      # calculate point 201's preheat
      pushtipforward2 = 0.012 - pushtipforward + deepchambumpmm # 12 mm forward to clear the existing extrudant (but still have the extrudant from this extrusion join the existing). subtract from previous to make it constant even if you change pushtipforward1
      preheatdistance = 0.010 # 10 mm . above what it would be pushed down
      point201a = p[p201x, p201y, z + preheatdistance, rx, ry, rz]
      p201bx = p201x + l1delxunit * pushtipforward2
      p201by = p201y + l1delyunit * pushtipforward2
      point201b = p[p201bx, p201by, z + preheatdistance, rx, ry, rz]
      point201c = p[p201bx, p201by, z, rx, ry, rz]

      # calculate point 202
      p202x = p201x + wd3 * l1delxunit
      p202y = p201y + wd3 * l1delyunit
      point202 = p[p202x, p202y, z, rx, ry, rz]

      struct2 = struct(point1=point1, point2=point2, point3=point3, point4=point4, point5=point5, point201=point201, point202=point202, point201a=point201a, point201b=point201b, point201c=point201c, point2a=point2a, point101=point101, point102=point102, point103=point103)
      return struct2
  end

  def calculate_LtAD_points_cover_left(struct1, leftwallthick, rightwallthick, deepcovercham):
      # get the stuff from the struct
      pointintersect = struct1[0]
      x0 = pointintersect[0]
      y0 = pointintersect[1]
      z0 = pointintersect[2]
      heading1 = struct1[1]
      heading2 = struct1[2]
      heading3 = struct1[3]
      l1delxunit = struct1[4]
      l1delyunit = struct1[5]
      l2delxunit = struct1[6]
      l2delyunit = struct1[7]

      # CONST
      welddistance1 = 6 # first path first leg (left side of L)
      welddistance2 = 6 # first path second leg (Right Side of L) # inches
      welddistance3 = 3 # second path (down sidewall) # inches

      wd1 = welddistance1 * 25.4 / 1000
      wd2 = welddistance2 * 25.4 / 1000
      wd3 = welddistance3 * 25.4 / 1000
      leftwallthickmm = leftwallthick * 25.4 / 1000 # in this step corner right, this is distance from left edge
      rightwallthickmm =  rightwallthick * 25.4 / 1000 # in this step corner right, this is distance from right edge

      if deepcovercham:
          deepchambumpmm = 0.09 * 25.4/1000 # if there is a deep chamfer on the cover, bump the welder inwards 0.09 more inches.
      else:
          deepchambumpmm = 0.0
      end

      # first, check if we need a lift column raise
      # (we do, because for maximum reach we want to make the lift pedestal be even with the top of the covers)
      zpi = pointintersect[2]
      if zpi > 0:
          liftcolumnzneeded = zpi * 1000.0 # the robot uses coordinates in meters, but the lift column uses coordinates in mm
          z0 = 0
      else:
          z0 = zpi
      end

      # first and second path

      # calculate rxryrz1 (facing down, preheat rightish)
      # start with rxryrz = 0,0,0 (gun facing up, preheat facing y+ axis)
      # rotate it 180 degrees about x axis. gun facing down, preheat facing y- axis
      # rotate it about 135 degrees ccw about z axis. x+ to heading3 is about 225 degrees. so our angle is heading3 - 90 degrees
      m1 = get_rotation_matrix_from_description("x", -1, 180 * pi / 180) # rotation 1: 180 degrees forward about x axis
      m2 = get_rotation_matrix_from_description("z", 1, heading3 - pi/2) # rotation 2
      m3 = multiply_matrix(m2, m1) #we rotate m1 first then m2, so we multiply in backwards order: 2 then 1
      rxryrz1 = convert_matrix_to_axang(m3)
      rx1 = rxryrz1[0]
      ry1 = rxryrz1[1]
      rz1 = rxryrz1[2]

      # calculate rxryrz2 (gun facing down, preheat facing right and back)
      # rotate 180 degrees about x. then rotate (90 deg + heading1 degrees) about z ccw
      m1 = get_rotation_matrix_from_description("x", -1, 180 * pi / 180)
      m2 = get_rotation_matrix_from_description("z", 1, heading1 + pi/2)
      m3 = multiply_matrix(m2, m1) #we rotate m1 first then m2, so we multiply in backwards order: 2 then 1
      rxryrz2 = convert_matrix_to_axang(m3)
      rx2 = rxryrz2[0]
      ry2 = rxryrz2[1]
      rz2 = rxryrz2[2]

      # calculate point centerchamfers (where the center of the two chamfers intersect
      pcx = x0 + (leftwallthickmm + deepchambumpmm) * l1delxunit + (rightwallthickmm + deepchambumpmm) * l2delxunit
      pcy = y0 + (leftwallthickmm + deepchambumpmm) * l1delyunit + (rightwallthickmm + deepchambumpmm) * l2delyunit
      pcz = z0

      # calculate point1 (start of weld)
      p1x = pcx + l2delxunit * wd1
      p1y = pcy + l2delyunit * wd1
      p1z = pcz
      point1 = p[p1x, p1y, p1z, rx1, ry1, rz1]

      # calculate point2 (end of segment 1)
      p2x = pcx
      p2y = pcy
      p2z = pcz
      point2 = p[p2x, p2y, p2z, rx1, ry1, rz1]

      # calculate point3 (point at end of turn)
      slide = 0.00 # slide distance : the distance the tip slides forward as it turns
      p3x = pcx + slide * l1delxunit
      p3y = pcy + slide * l1delyunit
      p3z = pcz
      point3 = p[p3x, p3y, p3z, rx2, ry2, rz2]

      # calculate point4 (end of segment 2)
      p4x = pcx + wd2 * l1delxunit
      p4y = pcy + wd2 * l1delyunit
      p4z = pcz
      point4 = p[p4x, p4y, p4z, rx2, ry2, rz2]

      # third path

      # calculate rxryrz3 (gun pointing down, preheat pointing toward corner. for left seam, pointing left)
      # start with rxryrz = 0,0,0 (gun facing up, preheat facing y+ axis.
      # rotate it 180 degrees about x axis. gun facing down, preheat facing y- axis
      # rotate it about 45 degrees ccw about z axis. x+ to heading1 is about 135 degrees. so our angle is heading1 - 90 degrees
      m1 = get_rotation_matrix_from_description("x", -1, 180 * pi / 180) # rotation 1: 180 degrees forward about x axis
      m2 = get_rotation_matrix_from_description("z", 1, heading1 - pi/2) # rotation 2
      m3 = multiply_matrix(m2, m1) #we rotate m1 first then m2, so we multiply in backwards order: 2 then 1
      rxryrz3 = convert_matrix_to_axang(m3)
      rx3 = rxryrz3[0]
      ry3 = rxryrz3[1]
      rz3 = rxryrz3[2]

      # calculate rxryrz4 (gun at 45 around corner)
      m1 = get_rotation_matrix_from_description("x", -1, 135 * pi / 180) # rotation 1: 135 degrees forward about x axis
      m2 = get_rotation_matrix_from_description("z", 1, heading1 - pi/2)
      m3 = multiply_matrix(m2, m1) #we rotate m1 first then m2, so we multiply in backwards order: 2 then 1
      rxryrz4 = convert_matrix_to_axang(m3)
      rx4 = rxryrz4[0]
      ry4 = rxryrz4[1]
      rz4 = rxryrz4[2]

      # calculate rxryrz5 (gun straight into left seam side chamfer, preheat down)
      # rotate about x 90 (forward). then rotate about z ~ 45 (ccw)
      m1 = get_rotation_matrix_from_description("x", -1, 90 * pi / 180)
      m2 = get_rotation_matrix_from_description("z", 1, heading1 - pi/2)
      m3 = multiply_matrix(m2, m1) #we rotate m1 first then m2, so we multiply in backwards order: 2 then 1
      rxryrz5 = convert_matrix_to_axang(m3)
      rx5 = rxryrz5[0]
      ry5 = rxryrz5[1]
      rz5 = rxryrz5[2]

      # calculate pointtopcham (the point at the top of the endwall chamfer) ( WHERE POINT3 WOULD BE IF RADIUS WAS 0)
      ptcx = x0 + rightwallthickmm * l2delxunit
      ptcy = y0 + rightwallthickmm * l2delyunit
      ptcz = z0

      # calculate point201 (weld start)
      # if deepchamfer, just ignore that. because if its deep chamfer then it filled more as well. so the hot extrudant should be to the same spot (same distance from the pointtopcham) whether it's big weld or small weld
      adjust = 0.0 # if you want to move the start point further away from corner (positive, mm) or closer to corner
      p201x = x0 + rightwallthickmm * l2delxunit + leftwallthickmm * l1delxunit + adjust * l1delxunit
      p201y = y0 + rightwallthickmm * l2delyunit + leftwallthickmm * l1delyunit + adjust * l1delyunit
      p201z = z0
      point201 = p[p201x, p201y, p201z, rx3, ry3, rz3]

      # the round over distance is the distance from pointbottomvcham to point2 (which will be the same as distance to p4)
      roundoverdistance = 0.05
      rod = roundoverdistance * 25.4 / 1000

      # calculate point202 (start of roundover)
      p202x = ptcx + rod * l1delxunit
      p202y = ptcy + rod * l1delyunit
      p202z = z0
      point202 = p[p202x, p202y, p202z, rx3, ry3, rz3]

      # calculate point203 (middle of roundover)
      # we know that the angle is exactly 90 degrees
      delta = calc_rod_midpoint_90deg(rod)
      p203z = ptcz - delta
      p203x = ptcx + delta * l1delxunit
      p203y = ptcy + delta * l1delyunit
      point203 = p[p203x, p203y, p203z, rx4, ry4, rz4]

      # calculate point204 (end of roundover)
      point204 = p[ptcx, ptcy, ptcz - rod, rx5, ry5, rz5]

      # calculate trail out points (tilt back and ride)
      botvcham = wd3 # where is the bottom of the v chamfer (z distance from top corner)
      tcpdiff = 14 # mm. the difference between backofhole tcp and welder tcp (tip)
      # point101 will still use backofhole, but points 102 and 103 will use normal weld tip tcp
      # calculate point5a (point101) (start of tilt back) (start of unflatten)
      dist = 1.5 * 25.4/1000 + tcpdiff/1000 # distance from botvcham
      p101x = ptcx
      p101y = ptcy
      p101z = ptcz - wd3 + dist
      point101 = p[p101x, p101y, p101z, rx5, ry5, rz5]

      # calculate point5b (point 102) (end of unflatten)
      dist = 0.5 * 25.4 / 1000
      tiltraise = 0.006
      p102x = ptcx + l1delxunit * tiltraise * -1
      p102y = ptcy + l1delyunit * tiltraise * -1
      p102z = ptcz - wd3 + dist

      # calculate rxryrz
      tiltangledeg = 10 # ten degree angle of tilt
      m1 = get_rotation_matrix_from_description("x", -1, (90 + tiltangledeg) * pi / 180) # rotation 1: 135 degrees forward about x axis
      m2 = get_rotation_matrix_from_description("z", 1, heading1 - pi/2)
      m3 = multiply_matrix(m2, m1) #we rotate m1 first then m2, so we multiply in backwards order: 2 then 1
      rxryrz = convert_matrix_to_axang(m3)
      rx = rxryrz[0]
      ry = rxryrz[1]
      rz = rxryrz[2]
      point102 = p[p102x, p102y, p102z, rx, ry, rz]

      # calculate point 5c (point 103) (end of smear)
      dist = -2 * 25.4/1000
      point103 = p[p102x, p102y, ptcz - wd3 + dist, rx, ry, rz]

      # return
      struct2 = struct(point1=point1, point2=point2, point3=point3, point4=point4, point201=point201, point202=point202, point203=point203, point204=point204, point101=point101, point102=point102, point103=point103)
      return struct2


  end

  def calculate_LtAD_points_cover_right(struct1, leftwallthick, rightwallthick, deepcovercham):
      # get the stuff from the struct
      pointintersect = struct1[0]
      x0 = pointintersect[0]
      y0 = pointintersect[1]
      z0 = pointintersect[2]
      heading1 = struct1[1]
      heading2 = struct1[2]
      heading3 = struct1[3]
      l1delxunit = struct1[4]
      l1delyunit = struct1[5]
      l2delxunit = struct1[6]
      l2delyunit = struct1[7]

      # CONST
      welddistance1 = 6 # first path first leg (left side of L)
      welddistance2 = 6 # first path second leg (Right Side of L) # inches
      welddistance3 = 3 # second path (down sidewall) # inches

      wd1 = welddistance1 * 25.4 / 1000
      wd2 = welddistance2 * 25.4 / 1000
      wd3 = welddistance3 * 25.4 / 1000
      leftwallthickmm = leftwallthick * 25.4 / 1000 # in this step corner right, this is distance from left edge
      rightwallthickmm =  rightwallthick * 25.4 / 1000 # in this step corner right, this is distance from right edge

      if deepcovercham:
          deepchambumpmm = 0.09 * 25.4/1000 # if there is a deep chamfer on the cover, bump the welder inwards 0.09 more inches.
      else:
          deepchambumpmm = 0.0
      end

      # first, check if we need a lift column raise
      # (we do, because for maximum reach we want to make the lift pedestal be even with the top of the covers)
      zpi = pointintersect[2]
      if zpi > 0:
          liftcolumnzneeded = zpi * 1000.0 # the robot uses coordinates in meters, but the lift column uses coordinates in mm
          z0 = 0
      else:
          z0 = zpi
      end

      # first and second path

      # calculate rxryrz1 (facing down, preheat rightish)
      # start with rxryrz = 0,0,0 (gun facing up, preheat facing y+ axis)
      # rotate it 180 degrees about x axis. gun facing down, preheat facing y- axis
      # rotate it about 135 degrees ccw about z axis. x+ to heading3 is about 225 degrees. so our angle is heading3 - 90 degrees
      m1 = get_rotation_matrix_from_description("x", -1, 180 * pi / 180) # rotation 1: 180 degrees forward about x axis
      m2 = get_rotation_matrix_from_description("z", 1, heading3 - pi/2) # rotation 2
      m3 = multiply_matrix(m2, m1) #we rotate m1 first then m2, so we multiply in backwards order: 2 then 1
      rxryrz1 = convert_matrix_to_axang(m3)
      rx1 = rxryrz1[0]
      ry1 = rxryrz1[1]
      rz1 = rxryrz1[2]

      # calculate rxryrz2 (gun facing down, preheat facing right and back)
      # rotate 180 degrees about x. then rotate (90 deg + heading1 degrees) about z ccw
      m1 = get_rotation_matrix_from_description("x", -1, 180 * pi / 180)
      m2 = get_rotation_matrix_from_description("z", 1, heading1 + pi/2)
      m3 = multiply_matrix(m2, m1) #we rotate m1 first then m2, so we multiply in backwards order: 2 then 1
      rxryrz2 = convert_matrix_to_axang(m3)
      rx2 = rxryrz2[0]
      ry2 = rxryrz2[1]
      rz2 = rxryrz2[2]

      # calculate point centerchamfers (where the center of the two chamfers intersect
      pcx = x0 + (leftwallthickmm + deepchambumpmm) * l1delxunit + (rightwallthickmm + deepchambumpmm) * l2delxunit
      pcy = y0 + (leftwallthickmm + deepchambumpmm) * l1delyunit + (rightwallthickmm + deepchambumpmm) * l2delyunit
      pcz = z0

      # calculate point1 (start of weld)
      p1x = pcx + l2delxunit * wd1
      p1y = pcy + l2delyunit * wd1
      p1z = pcz
      point1 = p[p1x, p1y, p1z, rx1, ry1, rz1]

      # calculate point2 (end of segment 1)
      p2x = pcx
      p2y = pcy
      p2z = pcz
      point2 = p[p2x, p2y, p2z, rx1, ry1, rz1]

      # calculate point3 (point at end of turn)
      slide = 0.00 # slide distance : the distance the tip slides forward as it turns
      p3x = pcx + slide * l1delxunit
      p3y = pcy + slide * l1delyunit
      p3z = pcz
      point3 = p[p3x, p3y, p3z, rx2, ry2, rz2]

      # calculate point4 (end of segment 2)
      p4x = pcx + wd2 * l1delxunit
      p4y = pcy + wd2 * l1delyunit
      p4z = pcz
      point4 = p[p4x, p4y, p4z, rx2, ry2, rz2]

      # third path

      # calculate rxryrz3 (gun pointing down, preheat pointing toward corner. for right seam, pointing right)
      # start with rxryrz = 0,0,0 (gun facing up, preheat facing y+ axis.
      # rotate it 180 degrees about x axis. gun facing down, preheat facing y- axis
      # rotate it about 135 degrees ccw about z axis. x+ to heading3 is about 225 degrees. so our angle is heading3 - 90 degrees
      m1 = get_rotation_matrix_from_description("x", -1, 180 * pi / 180) # rotation 1: 180 degrees forward about x axis
      m2 = get_rotation_matrix_from_description("z", 1, heading3 - pi/2) # rotation 2
      m3 = multiply_matrix(m2, m1) #we rotate m1 first then m2, so we multiply in backwards order: 2 then 1
      rxryrz3 = convert_matrix_to_axang(m3)
      rx3 = rxryrz3[0]
      ry3 = rxryrz3[1]
      rz3 = rxryrz3[2]

      # calculate rxryrz4 (gun at 45 around corner)
      m1 = get_rotation_matrix_from_description("x", -1, 135 * pi / 180) # rotation 1: 135 degrees forward about x axis
      m2 = get_rotation_matrix_from_description("z", 1, heading3 - pi/2)
      m3 = multiply_matrix(m2, m1) #we rotate m1 first then m2, so we multiply in backwards order: 2 then 1
      rxryrz4 = convert_matrix_to_axang(m3)
      rx4 = rxryrz4[0]
      ry4 = rxryrz4[1]
      rz4 = rxryrz4[2]

      # calculate rxryrz5 (gun straight into right seam side chamfer, preheat down)
      # rotate about x 90 (forward). then rotate about z ~ 135 (ccw)
      m1 = get_rotation_matrix_from_description("x", -1, 90 * pi / 180)
      m2 = get_rotation_matrix_from_description("z", 1, heading3 - pi/2)
      m3 = multiply_matrix(m2, m1) #we rotate m1 first then m2, so we multiply in backwards order: 2 then 1
      rxryrz5 = convert_matrix_to_axang(m3)
      rx5 = rxryrz5[0]
      ry5 = rxryrz5[1]
      rz5 = rxryrz5[2]

      # calculate rxryrz6 (gun straight into right seam side chamfer, preheat down, 10 degrees tiltback)
      tiltangledeg = 10 # ten degree angle of tilt
      m1 = get_rotation_matrix_from_description("x", -1, (90 + tiltangledeg) * pi / 180) # rotation 1: 135 degrees forward about x axis
      m2 = get_rotation_matrix_from_description("z", 1, heading3 - pi/2)
      m3 = multiply_matrix(m2, m1) #we rotate m1 first then m2, so we multiply in backwards order: 2 then 1
      rxryrz6 = convert_matrix_to_axang(m3)
      rx6 = rxryrz6[0]
      ry6 = rxryrz6[1]
      rz6 = rxryrz6[2]

      # calculate pointtopcham (the point at the top of the endwall chamfer) ( WHERE POINT3 WOULD BE IF RADIUS WAS 0)
      ptcx = x0 + leftwallthickmm * l1delxunit
      ptcy = y0 + leftwallthickmm * l1delyunit
      ptcz = z0

      # calculate point201 (weld start)
      # if deepchamfer, just ignore that. because if its deep chamfer then it filled more as well. so the hot extrudant should be to the same spot (same distance from the pointtopcham) whether it's big weld or small weld
      adjust = 0.0 # if you want to move the start point further away from corner (positive, mm) or closer to corner
      p201x = x0 + rightwallthickmm * l2delxunit + leftwallthickmm * l1delxunit + adjust * l2delxunit
      p201y = y0 + rightwallthickmm * l2delyunit + leftwallthickmm * l1delyunit + adjust * l2delyunit
      p201z = z0
      point201 = p[p201x, p201y, p201z, rx3, ry3, rz3]

      # the round over distance is the distance from pointbottomvcham to point2 (which will be the same as distance to p4)
      roundoverdistance = 0.05
      rod = roundoverdistance * 25.4 / 1000

      # calculate point202 (start of roundover)
      p202x = ptcx + rod * l2delxunit
      p202y = ptcy + rod * l2delyunit
      p202z = z0
      point202 = p[p202x, p202y, p202z, rx3, ry3, rz3]

      # calculate point203 (middle of roundover)
      # we know that the angle is exactly 90 degrees
      delta = calc_rod_midpoint_90deg(rod)
      p203z = ptcz - delta
      p203x = ptcx + delta * l2delxunit
      p203y = ptcy + delta * l2delyunit
      point203 = p[p203x, p203y, p203z, rx4, ry4, rz4]

      # calculate point204 (end of roundover)
      point204 = p[ptcx, ptcy, ptcz - rod, rx5, ry5, rz5]

      # calculate trail out points (tilt back and ride)
      botvcham = wd3 # where is the bottom of the v chamfer (z distance from top corner)
      tcpdiff = 14 # mm. the difference between backofhole tcp and welder tcp (tip)
      # point101 will still use backofhole, but points 102 and 103 will use normal weld tip tcp
      # calculate point5a (point101) (start of tilt back) (start of unflatten)
      dist = 1.5 * 25.4/1000 + tcpdiff/1000 # distance from botvcham
      p101x = ptcx
      p101y = ptcy
      p101z = ptcz - wd3 + dist
      point101 = p[p101x, p101y, p101z, rx5, ry5, rz5]

      # calculate point5b (point 102) (end of unflatten)
      dist = 0.5 * 25.4 / 1000
      tiltraise = 0.006
      p102x = ptcx + l2delxunit * tiltraise * -1
      p102y = ptcy + l2delyunit * tiltraise * -1
      p102z = ptcz - wd3 + dist
      point102 = p[p102x, p102y, p102z, rx6, ry6, rz6]

      # calculate point 5c (point 103) (end of smear)
      dist = -2 * 25.4/1000
      point103 = p[p102x, p102y, ptcz - wd3 + dist, rx6, ry6, rz6]

      # return
      struct2 = struct(point1=point1, point2=point2, point3=point3, point4=point4, point201=point201, point202=point202, point203=point203, point204=point204, point101=point101, point102=point102, point103=point103)
      return struct2

  end


  def main_calculate_cover_straight(p11, p12, p21, p22, sidewallthick, leftpoint, rightpoint, deepcovercham):
      struct1 = analyze_touchpoints_only_cover_straight(p11, p12, p21, p22, leftpoint)
      struct2 = calculate_straight_points_cover(struct1, sidewallthick, leftpoint, rightpoint, deepcovercham)
      #struct2 = calculate_DOtA_points_left_extended(struct1, list1, chamferover, chamferup, tcp_pose_top)
      #struct3 = check_validity_left(struct1, struct2)
      return struct2

  end

  # calculates the line of intersection of the sidewall plane (assumed vertical) and the cover plane (assumed perpendicular to sidewall plane)
  # returns a struct containing point0 (point on the intersection line, same y as leftpoint) and 3 components of the unit vector left to right and 2 components of the other direction in 2d
  def analyze_touchpoints_only_cover_straight(p11, p12, p21, p22, leftpoint):
      # calculate slope of sidewall in x-y plane
      # get the raw points from the first line
      l1p1x=p11[0]
      l1p1y=p11[1]
      l1p2x=p12[0]
      l1p2y=p12[1]

      # equate the first line in 2d space
      ml1 = (l1p2y-l1p1y) / (l1p2x-l1p1x)

      # b = y - mx
      bl1 = l1p1y - ml1 * l1p1x

      # calculate the cover plane
      # if two planes are perpendicular, then their normal vectors must be perpendicular.
      # the first planes normal vector is n1, which is taken from the equation of the plane ax + by + cz = d -> <a, b, c>
      # the second plane's normal vector is perpendicular to all vectors contained in the plane
      # p21 to p22 is a vector v contained within plane 2.
      # n2 is normal to both n1 AND v. to achieve a vector that is normal to both, take the cross product

      # plane 1 (y = mx + b) -> (b = -mx +1y +0z)
      n1 = [-1 * ml1, 1, 0]

      # v=P2−P1=(x2−x1,y2−y1,z2−z1)
      v = [p21[0]-p22[0], p21[1]-p22[1], p21[2]-p22[2]]

      #v n2 = cross product of n1 and v
      n2x = n1[1]*v[2] - n1[2]*v[1]
      n2y = n1[2]*v[0] - n1[0]*v[2]
      n2z = n1[0]*v[1] - n1[1]*v[0]
      n2 = [n2x, n2y, n2z]

      # find the d of the second plane
      # n2x * x + n2y * y + n2z * z = d0
      d = n2x * p21[0] + n2y * p21[1] + n2z * p21[2]

      # find the intersection line of the two planes
      # find the direction vector of that line by taking the cross product of the normal vector of those two planes
      v3x = n1[1]*n2[2] - n1[2]*n2[1]
      v3y = n1[2]*n2[0] - n1[0]*n2[2]
      v3z = n1[0]*n2[1] - n1[1]*n2[0]
      v3 = [v3x, v3y, v3z]

      # normalize the vector so the magnitude is 1
      magnitude2 = v3x * v3x + v3y * v3y + v3z * v3z
      magnitude = sqrt(magnitude2)
      v3xunit = v3x/magnitude
      v3yunit = v3y/magnitude
      v3zunit = v3z/magnitude

      # make sure it is going the right way (from left to right). make sure the v3yunit is positive
      if v3yunit < 0:
          v3xunit = v3xunit * -1
          v3yunit = v3yunit * -1
          v3zunit = v3zunit * -1
      end

      # next we have to find a point on the line by setting one of the dimensions and solving the system of equations
      # i will pick the y value of the left teach point
      y = leftpoint[1]
      # plane 1: -ml1 * x + 1 * y + 0 * z = bl1
      # -ml1 * x = bl1 - y
      x = (bl1 - y)/ (-1 * ml1)
      # plane 2: d = n2x * x + n2y * y + n2z * z
      # (d - n2x * x - n2y * y) = n2z * z
      z = (d - n2x * x - n2y * y) / n2z

      # make point0 into a pose
      point0 = p[x, y, z, 0, 0, 0]

      # find heading of main line
      heading1 = convert_uv_to_heading(v3xunit, v3yunit)

      # make a unit vector perpendicular to this one in the xy plane pointing x -. will be used to move over the chamfer distance
      ml2 = -1 / ml1
      # y = ml2 * x + unknownB
      # vector = [1, ml2]
      mag2 = 1 + ml2 * ml2
      mag = sqrt(mag2)
      v4xunit = 1 / mag
      v4yunit = ml2 / mag
      # switch is to the x direction is negative
      v4xunit = -1 * v4xunit
      v4yunit = -1 * v4yunit

      ret = struct(point0=point0, v3xunit=v3xunit, v3yunit=v3yunit, v3zunit=v3zunit, heading1=heading1, v4xunit=v4xunit, v4yunit=v4yunit)
      return ret
  end

  def calculate_straight_points_cover(struct1, sidewallthick, leftpointteach, rightpointteach, deepcovercham):
      # get the stuff
      point0 = struct1[0]
      p0x = point0[0]
      p0y = point0[1]
      p0z = point0[2]
      v3xunit = struct1[1]
      v3yunit = struct1[2]
      v3zunit = struct1[3]
      heading1 = struct1[4]
      v4xunit = struct1[5]
      v4yunit = struct1[6]
      sidewallthick = sidewallthick
      lpy = leftpointteach[1]
      rpy = rightpointteach[1]

      # first, check if we need a lift column raise
      # (we do, because for maximum reach we want to make the lift pedestal be even with the top of the covers)
      zpi = p0z
      if zpi > 0:
          liftcolumnzneeded = zpi * 1000.0 # the robot uses coordinates in meters, but the lift column uses coordinates in mm
          coverz = 0
      else:
          coverz = zpi
      end

      if deepcovercham:
          deepchambumpmm = 0.09 * 25.4/1000 # if there is a deep chamfer on the cover, bump the welder inwards 0.09 more inches.
      else:
          deepchambumpmm = 0.0
      end

      # calculate pointtopvcham
      chamferover = sidewallthick * 25.4 / 1000.0 + deepchambumpmm
      tiltraise = 0.006 # 6 mm raise needed for the tip to clear the plane during tiltback
      x = p0x + v4xunit * chamferover
      y = p0y + v4yunit * chamferover
      z = coverz + tiltraise

      # calculate rxryrz for tilted back
      # 3 rotations to make this happen.
      # start point is straight up with the preheat pointed in the +y direction.
      # first rotation is 180 degrees about x direction. gun is now pointing straight down with preheat facing -y direction
      m1 = get_rotation_matrix_from_description("x", 1, 180 * pi / 180)
      # second rotation is a 10 degree turn about the x axis (negative direction)
      m2 = get_rotation_matrix_from_description("x", -1, 10 * pi / 180)
      # third rotation is about 180 degrees about the z axis. starting from the -y axis, go until you get to heading1. that will equal heading1 plus 90 degrees
      m3 = get_rotation_matrix_from_description("z", 1, pi/2 + heading1)
      # combine them by multiplying m3 * m2 * m1
      # matrix multiplication is not commutative but it IS associative, so you can do this whichever order
      m4 = multiply_matrix(m2, m1)
      m5 = multiply_matrix(m3, m4)
      rxryrzt = convert_matrix_to_axang(m5)
      rxt = rxryrzt[0]
      ryt = rxryrzt[1]
      rzt = rxryrzt[2]
      pointtopvcham = p[x, y, z, rxt, ryt, rzt]

      # calculate point1 (preheat)
      dist = -1 * 25.4 / 1000.0 # move back 1 inch from
      p1x = x + dist * v3xunit
      p1y = y + dist * v3yunit
      p1z = z + dist * v3zunit
      point1 = p[p1x, p1y, p1z, rxt, ryt, rzt]

      # calculate point2 (start of flatten)
      dist = 0.5 * 25.4 / 1000.0  # half an inch past the top of v chamfer
      p2x = x + dist * v3xunit
      p2y = y + dist * v3yunit
      p2z = z + dist * v3zunit
      point2 = p[p2x, p2y, p2z, rxt, ryt, rzt]

      # calculate rxryrz for nontilted
      # first rotation is 180 degrees about x direction. gun is now pointing straight down with preheat facing -y direction
      m1 = get_rotation_matrix_from_description("x", 1, 180 * pi / 180)
      # third rotation is about 180 degrees about the z axis. starting from the -y axis, go until you get to heading1. that will equal heading1 plus 90 degrees
      m3 = get_rotation_matrix_from_description("z", 1, pi/2 + heading1)
      m5 = multiply_matrix(m3, m1)
      rxryrz = convert_matrix_to_axang(m5)
      rx = rxryrz[0]
      ry = rxryrz[1]
      rz = rxryrz[2]

      # calculate point3 (end of flatten)
      dist = 1.5 * 25.4 / 1000.0  # 1.5 inches past top of v chamfer
      p3x = x + dist * v3xunit
      p3y = y + dist * v3yunit
      p3z = coverz + dist * v3zunit
      point3 = p[p3x, p3y, p3z, rx, ry, rz]

      # calculate distance between leftpoint and rightpoint
      # we have the y distance. we need to find the total distance.
      # the unit vector (v3) should have a magnitude of 1. that's what analyze_touchpoints_only_cover_straight() calculated.
      # so the total distance is y distance * 1 / v3yunit
      ydist = rpy - lpy
      totdist = ydist / v3yunit

      # calculate pointtopvcham2
      x2 = x + v3xunit * totdist
      y2 = y + v3yunit * totdist
      z2 = z + v3zunit * totdist

      # calculate point4 (start of unflatten)
      dist = -1.5 * 25.4 / 1000.0
      p4x = x2 + v3xunit * dist
      p4y = y2 + v3yunit * dist
      p4z = z2 + v3zunit * dist - tiltraise
      point4 = p[p4x, p4y, p4z, rx, ry, rz]

      # calculate point5 (end of unflatten)
      dist = -0.5 * 25.4 / 1000.0
      p5x = x2 + v3xunit * dist
      p5y = y2 + v3yunit * dist
      p5z = z2 + v3zunit * dist
      point5 = p[p5x, p5y, p5z, rxt, ryt, rzt]

      # calculate point6 (end of smear)
      dist = 2 * 25.4 / 1000.0
      p6x = x2 + v3xunit * dist
      p6y = y2 + v3yunit * dist
      p6z = z2 + v3zunit * dist
      point6 = p[p6x, p6y, p6z, rxt, ryt, rzt]


      # return struct
      ret = struct(pointtopvcham=pointtopvcham, point1=point1, point2=point2, point3=point3, point4=point4, point5=point5, point6=point6)
      return ret


  end

  def main_calculate_floor_straight(p11, p12, p21, p22, floorthick, leftpoint, rightpoint):
      struct1 = analyze_touchpoints_only_cover_straight(p11, p12, p21, p22, leftpoint)
      struct2 = calculate_straight_points_floor(struct1, floorthick, leftpoint, rightpoint)
      #struct2 = calculate_DOtA_points_left_extended(struct1, list1, chamferover, chamferup, tcp_pose_top)
      #struct3 = check_validity_left(struct1, struct2)
      return struct2

  end

  # the path for welding a floor straight weld with v chisels on both sides.
  # start at the right side and move left.
  def calculate_straight_points_floor(struct1, floorthick, leftpointteach, rightpointteach):
      # get the stuff
      point0 = struct1[0]
      p0x = point0[0]
      p0y = point0[1]
      p0z = point0[2]
      v3xunit = struct1[1]
      v3yunit = struct1[2]
      v3zunit = struct1[3]
      heading1 = struct1[4]
      v4xunit = struct1[5]
      v4yunit = struct1[6]
      lpy = leftpointteach[1]
      rpy = rightpointteach[1]

      # first, check if we need a lift column raise
      # (we do not, because the floors are low)
      zpi = p0z
      floorz = zpi

      # calculate pointtopvcham (left point) (tilted and tiltraised)
      chamferup = floorthick * 25.4 / 1000.0
      tiltraise = 0.006 # 6 mm raise needed for the tip to clear the plane during tiltback
      # on this one, move the tiltraise distance sideways (towards robot) and the chamferover distance up
      x = p0x + v4xunit * tiltraise * -1
      y = p0y + v4yunit * tiltraise * -1
      z = floorz + chamferup

      # calculate rxryrz for tilted back
      # 3 rotations to make this happen.
      # start point is straight up with the preheat pointed in the +y direction.
      # first rotation is 90 degrees about y axis. positive direction. gun is now pointing in the x+ direction with preheat facing +y direction
      m1 = get_rotation_matrix_from_description("y", 1, 90 * pi / 180)
      # second rotation is about 180 degrees about the z axis. heading1 plus 90 degrees. gun is now pointing directly into the sidewall
      m2 = get_rotation_matrix_from_description("z", 1, pi/2 + heading1)
      # third rotation is 10 degrees about the z axis. gun is now tilted back 10 degrees from the sidewall
      m3 = get_rotation_matrix_from_description("z", 1, 10 * pi / 180)
      # combine them by multiplying m3 * m2 * m1
      # matrix multiplication is not commutative but it IS associative, so you can do this whichever order
      m4 = multiply_matrix(m2, m1)
      m5 = multiply_matrix(m3, m4)
      rxryrzt = convert_matrix_to_axang(m5)
      rxt = rxryrzt[0]
      ryt = rxryrzt[1]
      rzt = rxryrzt[2]
      # the non tilted angle is just m4
      rxryrz = convert_matrix_to_axang(m4)
      rx = rxryrz[0]
      ry = rxryrz[1]
      rz = rxryrz[2]
      pointtopvcham = p[x, y, z, rxt, ryt, rzt]

      # calculate distance between leftpoint and rightpoint
      # we have the y distance. we need to find the total distance.
      # the unit vector (v3) should have a magnitude of 1. that's what analyze_touchpoints_only_cover_straight() calculated.
      # so the total distance is y distance * 1 / v3yunit
      ydist = rpy - lpy
      totdist = ydist / v3yunit

      # calculate pointtopvcham2 (right point) (tilted and tiltraised)
      x2 = x + v3xunit * totdist
      y2 = y + v3yunit * totdist
      z2 = z + v3zunit * totdist
      pointtopvcham2 = p[x2, y2, z2, rxt, ryt, rzt]

      # calculate point1 (preheat)
      dist = 1 * 25.4 / 1000.0 # move back 1 inch from ptvc2 (in this case back means positive)
      p1x = x2 + dist * v3xunit
      p1y = y2 + dist * v3yunit
      p1z = z2 + dist * v3zunit
      point1 = p[p1x, p1y, p1z, rxt, ryt, rzt]

      # calculate point2 (start of flatten)
      dist = -0.5 * 25.4 / 1000.0  # half an inch past the top of v chamfer
      p2x = x2 + dist * v3xunit
      p2y = y2 + dist * v3yunit
      p2z = z2 + dist * v3zunit
      point2 = p[p2x, p2y, p2z, rxt, ryt, rzt]

      # calculate point3 (end of flatten)
      dist = -1.5 * 25.4 / 1000.0  # 1.5 inches past top of v chamfer
      p3x = x2 + dist * v3xunit + tiltraise * v4xunit
      p3y = y2 + dist * v3yunit + tiltraise * v4yunit
      p3z = z2 + dist * v3zunit
      point3 = p[p3x, p3y, p3z, rx, ry, rz]

      # calculate point4 (start of unflatten)
      dist = 1.5 * 25.4 / 1000.0
      p4x = x + v3xunit * dist + tiltraise * v4xunit
      p4y = y + v3yunit * dist + tiltraise * v4yunit
      p4z = z + v3zunit * dist
      point4 = p[p4x, p4y, p4z, rx, ry, rz]

      # calculate point5 (end of unflatten)
      dist = 0.5 * 25.4 / 1000.0
      p5x = x + v3xunit * dist
      p5y = y + v3yunit * dist
      p5z = z + v3zunit * dist
      point5 = p[p5x, p5y, p5z, rxt, ryt, rzt]

      # calculate point6 (end of smear)
      dist = -2 * 25.4 / 1000.0
      p6x = x + v3xunit * dist
      p6y = y + v3yunit * dist
      p6z = z + v3zunit * dist
      point6 = p[p6x, p6y, p6z, rxt, ryt, rzt]

      # return struct
      ret = struct(pointtopvcham=pointtopvcham, point1=point1, point2=point2, point3=point3, point4=point4, point5=point5, point6=point6)
      return ret

  end

  # this function determines the starting touchpoints for homing in on cover lt geometry
  # includes two points above the cover lt, closer to the robot than the lt, facing down
  def get_coverlt_homing_pathpoints(leftpoint, rightpoint):
      # get the teach position points
      lpx = leftpoint[0]
      lpy = leftpoint[1]
      lpz = leftpoint[2]
      rpx = rightpoint[0]
      rpy = rightpoint[1]
      rpz = rightpoint[2]

      # specify the distances from (in meters)
      d0 = 0.05 # how far from the cover to approach from
      d1 = 0.03 # how far the touchpints are pushed closer to the robot
      d2 = 0.00 # how far inwards the touchpoints are pushed

      # rxryrz
      rxryrz = [0.334, 3.124, 0]
      rx = rxryrz[0]
      ry = rxryrz[1]
      rz = rxryrz[2]

      # calculate the points
      ph1 = p[lpx + d1, lpy + d2, lpz + d0, rx, ry, rz] # left side approach
      ph2 = p[rpx + d1, rpy - d2, rpz + d0, rx, ry, rz] # right side approach

      ret = struct(ph1=ph1, ph2=ph2)
      is_robot_at_reachable_spot(leftpoint, ret)
      return ret
  end

  def main_calculate_cover_lt(p11, p12, leftpoint, rightpoint):
      struct1 = analyze_touchpoints_only_cover_lt(p11, p12, leftpoint, rightpoint)
      struct2 = calculate_points_cover_lt(struct1)
      #struct2 = calculate_DOtA_points_left_extended(struct1, list1, chamferover, chamferup, tcp_pose_top)
      #struct3 = check_validity_left(struct1, struct2)
      return struct2

  end

  def analyze_touchpoints_only_cover_lt(p11, p12, leftpoint, rightpoint):
      # calculate the slope of the groove in xy plane
      l1p1x = leftpoint[0]
      l1p1y = leftpoint[1]
      l1p2x = rightpoint[0]
      l1p2y = rightpoint[1]

      # equate the first line in 2d space
      ml1 = (l1p2y-l1p1y) / (l1p2x-l1p1x)

      # b = y - mx
      bl1 = l1p1y - ml1 * l1p1x

      # zraise (how much the z value changes from left point to right point
      zraise = p12[2] - p11[2]

      #get the calcpoints
      leftcalcpoint = [leftpoint[0], leftpoint[1], p11[2]]
      rightcalcpoint = [rightpoint[0], rightpoint[1], p12[2]]
      # get the vector from a to b
      vec = [rightcalcpoint[0] - leftcalcpoint[0], rightcalcpoint[1] - leftcalcpoint[1], rightcalcpoint[2] - leftcalcpoint[2]]
      # get the unit vector in 3d
      mag3d = sqrt(vec[0]*vec[0]+vec[1]*vec[1]+vec[2]*vec[2])
      vec3dunit = [vec[0]/mag3d, vec[1]/mag3d, vec[2]/mag3d]
      # get the unit vector in 2d
      mag2d = sqrt(vec[0]*vec[0]+vec[1]*vec[1])
      vec2dunit = [vec[0]/mag2d, vec[1]/mag2d]
      # get the heading
      heading1 = convert_uv_to_heading(vec2dunit[0], vec2dunit[1])

      ret = struct(leftcalcpoint=leftcalcpoint, rightcalcpoint=rightcalcpoint, vxunit=vec3dunit[0], vyunit=vec3dunit[1], vzunit=vec3dunit[2], heading1=heading1)
      return ret
  end

  def calculate_points_cover_lt(struct1):
      # get the stuff from struct
      leftcalcpoint = struct1[0]
      x = leftcalcpoint[0]
      y = leftcalcpoint[1]
      z = leftcalcpoint[2]
      rightcalcpoint = struct1[1]
      x2 = rightcalcpoint[0]
      y2 = rightcalcpoint[1]
      z2 = rightcalcpoint[2]
      v3xunit = struct1[2]
      v3yunit = struct1[3]
      v3zunit = struct1[4]
      heading1 = struct1[5]

      # first calculate rxryrz f normal and tiltback
      # calculate rxryrz for tilted back
      # 3 rotations to make this happen.
      # start point is straight up with the preheat pointed in the +y direction.
      # first rotation is 180 degrees about x direction. gun is now pointing straight down with preheat facing -y direction
      m1 = get_rotation_matrix_from_description("x", 1, 180 * pi / 180)
      # second rotation is a 10 degree turn about the x axis (negative direction)
      m2 = get_rotation_matrix_from_description("x", -1, 10 * pi / 180)
      # third rotation is about 180 degrees about the z axis. starting from the -y axis, go until you get to heading1. that will equal heading1 plus 90 degrees
      m3 = get_rotation_matrix_from_description("z", 1, pi/2 + heading1)
      # combine them by multiplying m3 * m2 * m1
      # matrix multiplication is not commutative but it IS associative, so you can do this whichever order
      m4 = multiply_matrix(m2, m1)
      m5 = multiply_matrix(m3, m4)
      rxryrzt = convert_matrix_to_axang(m5)
      rxt = rxryrzt[0]
      ryt = rxryrzt[1]
      rzt = rxryrzt[2]

      # calculate rxryrz for nontilted
      # first rotation is 180 degrees about x direction. gun is now pointing straight down with preheat facing -y direction
      m1 = get_rotation_matrix_from_description("x", 1, 180 * pi / 180)
      # third rotation is about 180 degrees about the z axis. starting from the -y axis, go until you get to heading1. that will equal heading1 plus 90 degrees
      m3 = get_rotation_matrix_from_description("z", 1, pi/2 + heading1)
      m5 = multiply_matrix(m3, m1)
      rxryrz = convert_matrix_to_axang(m5)
      rx = rxryrz[0]
      ry = rxryrz[1]
      rz = rxryrz[2]

      tiltraise = 0.006 # 6 mm raise needed for the tip to clear the plane during tiltback

      # calculate points 1-3
      # calculate point1 (preheat)
      dist = -1 * 25.4 / 1000.0 # move back 1 inch from
      p1x = x + dist * v3xunit
      p1y = y + dist * v3yunit
      p1z = z + dist * v3zunit + tiltraise
      point1 = p[p1x, p1y, p1z, rxt, ryt, rzt]

      # calculate point2 (start of flatten)
      dist = 0.5 * 25.4 / 1000.0  # half an inch past the top of v chamfer
      p2x = x + dist * v3xunit
      p2y = y + dist * v3yunit
      p2z = z + dist * v3zunit + tiltraise
      point2 = p[p2x, p2y, p2z, rxt, ryt, rzt]

      # calculate point3 (end of flatten)
      dist = 1.5 * 25.4 / 1000.0  # 1.5 inches past top of v chamfer
      p3x = x + dist * v3xunit
      p3y = y + dist * v3yunit
      p3z = z + dist * v3zunit
      point3 = p[p3x, p3y, p3z, rx, ry, rz]

      # calculate points 4-6
      # calculate point4 (start of unflatten)
      dist = -1.5 * 25.4 / 1000.0
      p4x = x2 + v3xunit * dist
      p4y = y2 + v3yunit * dist
      p4z = z2 + v3zunit * dist
      point4 = p[p4x, p4y, p4z, rx, ry, rz]

      # calculate point5 (end of unflatten)
      dist = -0.5 * 25.4 / 1000.0
      p5x = x2 + v3xunit * dist
      p5y = y2 + v3yunit * dist
      p5z = z2 + v3zunit * dist + tiltraise
      point5 = p[p5x, p5y, p5z, rxt, ryt, rzt]

      # calculate point6 (end of smear)
      dist = 2 * 25.4 / 1000.0
      p6x = x2 + v3xunit * dist
      p6y = y2 + v3yunit * dist
      p6z = z2 + v3zunit * dist + tiltraise
      point6 = p[p6x, p6y, p6z, rxt, ryt, rzt]

      # return struct
      ret = struct(pointtopvcham=leftcalcpoint, point1=point1, point2=point2, point3=point3, point4=point4, point5=point5, point6=point6)
      return ret

  end

  def main_calculate_sleeve_fillet(p1, p2, p3):
      struct1 = analyze_touchpoints_only_sleeve_fillet(p1, p2, p3)
      struct2 = calculate_points_sleeve_fillet(struct1)
      return struct2
  end

  # given 3 points at the intersection of the sleeve and the sidewall, this calculates and returns 3 things:
  # the centerpoint of the circle on the plane, the normal vector of the plane, and the radius of the circle
  # then it returns 4 more things after converting to a vertical circle/plane: heading1 (into the plane), vecn, vecr, vecu
  def analyze_touchpoints_only_sleeve_fillet(p1, p2, p3):
      x1 = p1[0]
      y1 = p1[1]
      z1 = p1[2]
      x2 = p2[0]
      y2 = p2[1]
      z2 = p2[2]
      x3 = p3[0]
      y3 = p3[1]
      z3 = p3[2]

      # calculate plane
      # calculate ab (1->2) vector
      abvec = [x2-x1, y2-y1, z2-z1]
      # calculate ac (1->3) vector
      acvec = [x3-x1, y3-y1, z3-z1]
      #calculate the plane's normal vector = ab x ac

      n = crossproduct(abvec, acvec)
      mag = sqrt(n[0]*n[0]+n[1]*n[1]+n[2]*n[2])
      n = [n[0]/mag, n[1]/mag, n[2]/mag]
      d = n[0] * x1 + n[1] * y1 + n[2] * z1

      # find the circle
      # Midpoint of AB:
      mab = [(x1 + x2)/2, (y1 + y2)/2, (z1 + z2)/2]
      # midpoint of ac
      mac = [(x3 + x1)/2, (y3 + y1)/2, (z3 + z1)/2]
      # Get Normal Vectors to AB and AC in the Plane
      # nab (normal to ab) = abvec x n
      nab = crossproduct(abvec, n)
      # nac (normal to ac) = acvec x n
      nac = crossproduct(acvec, n)
      # Define Perpendicular Bisector Lines
      # Each line goes through a midpoint and extends in the direction of the na_
      # we already have the equations of those lines in point vector form with l1 = mab + s * nab, and l2 = mac + t * nac
      # define all the terms so the math is simpler when i have to do math
      mabx = mab[0]
      maby = mab[1]
      mabz = mab[2]
      nabx = nab[0]
      naby = nab[1]
      nabz = nab[2]
      macx = mac[0]
      macy = mac[1]
      macz = mac[2]
      nacx = nac[0]
      nacy = nac[1]
      nacz = nac[2]
      # find the intersection point using the y and z equations
      # maby + s * naby = macy + t * nacy
      # mabz + s * nabz = macz + t * nacz
      # first solve for s and take
      # t = (macz*naby + maby*nabz - mabz*naby - macy*nabz) / (nacy*nabz - naby*nacz)
      t = (macz*naby + maby*nabz - mabz*naby - macy*nabz) / (nacy*nabz - naby*nacz)
      # s = (t*nacz + macz - mabz) / nabz
      s = (t*nacz + macz - mabz) / nabz
      # find the point
      # pcenter = mac + t * nac
      pcenterx = macx + t * nacx
      pcentery = macy + t * nacy
      pcenterz = macz + t * nacz
      rxryrz = [0.528, 4.631, 0.258] # demo point of the welder pointing forward into a sleeve
      pcenter = p[pcenterx, pcentery, pcenterz, rxryrz[0], rxryrz[1], rxryrz[2]]
      radius = distance_between(pcenterx, pcentery, pcenterz, x1, y1, z1)

      # ------ start calculation of vertical assumption -----
      # assume the plane close to vertical
      # fix it to make it actually vertical
      # calculate the unit vector of up, and the unit vector of right.
      # calculate the heading from the +x axis to pointing straight into the wall.
      # the unit vector of up is [0, 0, 1] (because the plane is verticalized) (for easier calculations)
      # first calculate the normal vector INTO the sidewall (make sure x is negative) and make it a unit vector
      vecn = [n[0], n[1], 0] # vector normal
      if vecn[0] > 0:
          vecn = [-n[0], -n[1], 0]
      end
      mag = sqrt(vecn[0]*vecn[0]+vecn[1]*vecn[1])
      vecn = [vecn[0]/mag, vecn[1]/mag, 0]
      # next calculate the right normal vector (the vector IN the plane that goes to the right)
      vecr = [vecn[1], -1*vecn[0], 0]
      vecu = [0, 0, 1] # vector up
      heading1 = convert_uv_to_heading(vecn[0], vecn[1])


      ret = struct(pcenter=pcenter, planenormalvec=n, radius=radius, heading1=heading1, vecn=vecn, vecr=vecr, vecu=vecu)
      return ret
  end

  def crossproduct(vec1, vec2):
      nx = vec1[1]*vec2[2] - vec1[2]*vec2[1]
      ny = vec1[2]*vec2[0] - vec1[0]*vec2[2]
      nz = vec1[0]*vec2[1] - vec1[1]*vec2[0]
      ret = [nx, ny, nz]
      return ret
  end

  # this function calculates only the four points of the quadrants, for the not real program.
  # these calculations are easier so that's why i'm starting with them first.
  # this assumes a vertical plane
  def calculate_points_sleeve_fillet_quadonly(struct1):
      # get the stuff from the struct
      pcenter = struct1[0]
      pcx = pcenter[0]
      pcy = pcenter[1]
      pcz = pcenter[2]
      planenormalvec = struct1[1]
      radius = struct1[2]
      heading1 = struct1[3]
      vecn = struct1[4]
      vecnx = vecn[0]
      vecny = vecn[1]
      vecr = struct1[5]
      vecrx = vecr[0]
      vecry = vecr[1]
      vecu = struct1[6]
      vecuz = vecu[2]

      # define cushions (the backofhole can't actually touch the intersection of pipe and wall, it travels a certain distance around it
      cushout = 0.006 # 5mm # the cushion out from the wall
      cusharound = 0.006 # 5mm # the cushion around the sleeve.

      # get the top point (point1)
      # take the center point and move up the radius plus the cushions
      p1x = pcx + vecnx * -1 * cushout
      p1y = pcy + vecny * -1 * cushout
      p1z = pcz + vecuz * radius + vecuz * cusharound

      # find rxryrz1
      # first rotation is 135 degrees about the y- direction. 90 degrees to get flat. Tip pointing x-, preheat pointing y+. 45 more degrees to get at that above angle
      m1 = get_rotation_matrix_from_description("y", -1, 135 * pi / 180)
      # second rotation is heading1 – 180 degrees about the z+ axis to get pointing straight into wall. Heading1 should be about 180 degrees
      m2 = get_rotation_matrix_from_description("z", 1, heading1 - 180 * pi/180)
      # combine them by multiplying
      m3 = multiply_matrix(m2, m1)
      rxryrz1 = convert_matrix_to_axang(m3)
      rx1 = rxryrz1[0]
      ry1 = rxryrz1[1]
      rz1 = rxryrz1[2]

      point1 = p[p1x, p1y, p1z, rx1, ry1, rz1]

      # get second point (right) (point2)
      # take the center point and move right the radius plus the cushions
      p2x = pcx + vecrx * radius + vecrx * cusharound + vecnx * -1 * cushout
      p2y = pcy + vecry * radius + vecry * cusharound + vecny * -1 * cushout
      p2z = pcz

      # find rxryrz2
      # first rotation is 90 degrees about the x- axis
      m1 = get_rotation_matrix_from_description("x", -1, 90 * pi / 180)
      # second rotation is About 135 degrees about the z+ axis. This calculation is heading1 – 45 degrees
      m2 = get_rotation_matrix_from_description("z", 1, heading1 - 45 * pi/180)
      # combine them by multiplying
      m3 = multiply_matrix(m2, m1)
      rxryrz2 = convert_matrix_to_axang(m3)
      rx2 = rxryrz2[0]
      ry2 = rxryrz2[1]
      rz2 = rxryrz2[2]

      point2 = p[p2x, p2y, p2z, rx2, ry2, rz2]

      # get the third point (bottom) (point3)
      p3x = pcx + vecnx * -1 * cushout
      p3y = pcy + vecny * -1 * cushout
      p3z = pcz - vecuz * radius - vecuz * cusharound

      # find rxryrz3
      # first rotation is 45 degrees about the y+ axis
      m1 = get_rotation_matrix_from_description("y", 1, 45 * pi / 180)
      # second rotation is About 180 degrees about the z+ axis. This calculation is heading1 degrees
      m2 = get_rotation_matrix_from_description("z", 1, heading1)
      # combine them by multiplying
      m3 = multiply_matrix(m2, m1)
      rxryrz3 = convert_matrix_to_axang(m3)
      rx3 = rxryrz3[0]
      ry3 = rxryrz3[1]
      rz3 = rxryrz3[2]

      point3 = p[p3x, p3y, p3z, rx3, ry3, rz3]

      # get the fourth point (left) (point4)
      p4x = pcx - vecrx * radius - vecrx * cusharound + vecnx * -1 * cushout
      p4y = pcy - vecry * radius - vecry * cusharound + vecny * -1 * cushout
      p4z = pcz

      # find rxryrz4
      # first rotation is 90 degrees about the x+ axis
      m1 = get_rotation_matrix_from_description("x", 1, 90 * pi / 180)
      # second rotation is heading1 + 45 degrees about the z+ axis. approx 225 degrees ccw
      m2 = get_rotation_matrix_from_description("z", 1, heading1 + 45 * pi/180)
      # combine them by multiplying
      m3 = multiply_matrix(m2, m1)
      rxryrz4 = convert_matrix_to_axang(m3)
      rx4 = rxryrz4[0]
      ry4 = rxryrz4[1]
      rz4 = rxryrz4[2]

      point4 = p[p4x, p4y, p4z, rx4, ry4, rz4]

      # return the points
      ret = struct(point1=point1, point2=point2, point3=point3, point4=point4)
      return ret

  end

  # this function calculates the points necessary for the fillet sleeve weld path.
  # this assumes a vertical plane
  def calculate_points_sleeve_fillet(struct1):
      # get the stuff from the struct
      pcenter = struct1[0]
      pcx = pcenter[0]
      pcy = pcenter[1]
      pcz = pcenter[2]
      planenormalvec = struct1[1]
      radius = struct1[2]
      heading1 = struct1[3]
      vecn = struct1[4]
      vecnx = vecn[0]
      vecny = vecn[1]
      vecr = struct1[5]
      vecrx = vecr[0]
      vecry = vecr[1]
      vecu = struct1[6]
      vecuz = vecu[2]

      # define cushions (the backofhole can't actually touch the intersection of pipe and wall, it travels a certain distance around it
      cushout = 0.006 # 5mm # the cushion out from the wall
      cusharound = 0.004 # 5mm # the cushion around the sleeve.

      # get the top point (point1)
      # take the center point and move up the radius plus the cushions
      p1x = pcx + vecnx * -1 * cushout
      p1y = pcy + vecny * -1 * cushout
      p1z = pcz + vecuz * radius + vecuz * cusharound

      # find rxryrz1
      # first rotation is 135 degrees about the y- direction. 90 degrees to get flat. Tip pointing x-, preheat pointing y+. 45 more degrees to get at that above angle
      m1 = get_rotation_matrix_from_description("y", -1, 135 * pi / 180)
      # second rotation is heading1 – 180 degrees about the z+ axis to get pointing straight into wall. Heading1 should be about 180 degrees
      m2 = get_rotation_matrix_from_description("z", 1, heading1 - 180 * pi/180)
      # combine them by multiplying
      m3 = multiply_matrix(m2, m1)
      rxryrz1 = convert_matrix_to_axang(m3)
      rx1 = rxryrz1[0]
      ry1 = rxryrz1[1]
      rz1 = rxryrz1[2]

      point1 = p[p1x, p1y, p1z, rx1, ry1, rz1]

      # get second point (right) (point2)
      # take the center point and move right the radius plus the cushions
      p2x = pcx + vecrx * radius + vecrx * cusharound + vecnx * -1 * cushout
      p2y = pcy + vecry * radius + vecry * cusharound + vecny * -1 * cushout
      p2z = pcz

      # find rxryrz2
      # first rotation is 90 degrees about the x- axis
      m1 = get_rotation_matrix_from_description("x", -1, 90 * pi / 180)
      # second rotation is About 135 degrees about the z+ axis. This calculation is heading1 – 45 degrees
      m2 = get_rotation_matrix_from_description("z", 1, heading1 - 45 * pi/180)
      # combine them by multiplying
      m3 = multiply_matrix(m2, m1)
      rxryrz2 = convert_matrix_to_axang(m3)
      rx2 = rxryrz2[0]
      ry2 = rxryrz2[1]
      rz2 = rxryrz2[2]

      point2 = p[p2x, p2y, p2z, rx2, ry2, rz2]

      # get the third point (bottom) (point3)
      p3x = pcx + vecnx * -1 * cushout
      p3y = pcy + vecny * -1 * cushout
      p3z = pcz - vecuz * radius - vecuz * cusharound

      # find rxryrz3
      # first rotation is 45 degrees about the y+ axis
      m1 = get_rotation_matrix_from_description("y", 1, 45 * pi / 180)
      # second rotation is About 180 degrees about the z+ axis. This calculation is heading1 degrees
      m2 = get_rotation_matrix_from_description("z", 1, heading1)
      # combine them by multiplying
      m3 = multiply_matrix(m2, m1)
      rxryrz3 = convert_matrix_to_axang(m3)
      rx3 = rxryrz3[0]
      ry3 = rxryrz3[1]
      rz3 = rxryrz3[2]

      point3 = p[p3x, p3y, p3z, rx3, ry3, rz3]

      # get the fourth point (left) (point4)
      p4x = pcx - vecrx * radius - vecrx * cusharound + vecnx * -1 * cushout
      p4y = pcy - vecry * radius - vecry * cusharound + vecny * -1 * cushout
      p4z = pcz

      # find rxryrz4
      # first rotation is 90 degrees about the x+ axis
      m1 = get_rotation_matrix_from_description("x", 1, 90 * pi / 180)
      # second rotation is heading1 + 45 degrees about the z+ axis. approx 225 degrees ccw
      m2 = get_rotation_matrix_from_description("z", 1, heading1 + 45 * pi/180)
      # combine them by multiplying
      m3 = multiply_matrix(m2, m1)
      rxryrz4 = convert_matrix_to_axang(m3)
      rx4 = rxryrz4[0]
      ry4 = rxryrz4[1]
      rz4 = rxryrz4[2]

      point4 = p[p4x, p4y, p4z, rx4, ry4, rz4]

      # get the angle for the tilt-back at the top (p1)
      m0 = get_rotation_matrix_from_description("x", -1, 10 * pi / 180)
      m1 = get_rotation_matrix_from_description("y", -1, 135 * pi / 180)
      # second rotation is heading1 – 180 degrees about the z+ axis to get pointing straight into wall. Heading1 should be about 180 degrees
      m2 = get_rotation_matrix_from_description("z", 1, heading1 - 180 * pi/180)
      # combine them by multiplying
      m3 = multiply_matrix(m2, m1)
      m4 = multiply_matrix(m3, m0)
      rxryrz1tilt = convert_matrix_to_axang(m4)
      rx1t = rxryrz1tilt[0]
      ry1t = rxryrz1tilt[1]
      rz1t = rxryrz1tilt[2]

      # point 1, but with the tilt back angle
      point1t = p[p1x, p1y, p1z, rx1t, ry1t, rz1t]

      # point45 (the point 45 degrees along the path) (has no rxryrz data) (because if we do fixed angle circle move it wont use that anyways, it'l just use the angle from p1t)
      distup = cos(45 * pi/180) * (radius + cusharound)
      distover = sin(45 * pi/180) * (radius + cusharound)
      p45x = pcx + vecrx * distover + vecnx * -1 * cushout
      p45y = pcy + vecry * distover + vecny * -1 * cushout
      p45z = pcz + vecuz * distup
      point45 = p[p45x, p45y, p45z, 0,0,0]

      # point22 (22.5 degrees of angle)
      distup = cos(22.5 * pi/180) * (radius + cusharound)
      distover = sin(22.5 * pi/180) * (radius + cusharound)
      p22x = pcx + vecrx * distover + vecnx * -1 * cushout
      p22y = pcy + vecry * distover + vecny * -1 * cushout
      p22z = pcz + vecuz * distup
      point22 = p[p22x, p22y, p22z, 0,0,0]

      # return the points
      ret = struct(point1=point1, point2=point2, point3=point3, point4=point4, point1t=point1t, point45=point45, point22=point22)
      return ret

  end

  def make_pose_list(length):
      if length < 1:
          ret = []
          return ret
      end
      if length == 1:
          pose_list = [p[0, 0, 0, 0, 0, 0]]
          return pose_list
      end
      if length == 2:
          pose_list = [p[0, 0, 0, 0, 0, 0], p[0, 0, 0, 0, 0, 0]]
          return pose_list
      end
      if length == 3:
          pose_list = [p[0, 0, 0, 0, 0, 0], p[0, 0, 0, 0, 0, 0], p[0, 0, 0, 0, 0, 0]]
          return pose_list
      end
      if length == 4:
          pose_list = [p[0, 0, 0, 0, 0, 0], p[0, 0, 0, 0, 0, 0], p[0, 0, 0, 0, 0, 0], p[0, 0, 0, 0, 0, 0]]
          return pose_list
      end
      if length == 5:
          pose_list = [p[0, 0, 0, 0, 0, 0], p[0, 0, 0, 0, 0, 0], p[0, 0, 0, 0, 0, 0], p[0, 0, 0, 0, 0, 0], p[0, 0, 0, 0, 0, 0]]
          return pose_list
      end
      if length == 6:
          pose_list = [p[0, 0, 0, 0, 0, 0], p[0, 0, 0, 0, 0, 0], p[0, 0, 0, 0, 0, 0], p[0, 0, 0, 0, 0, 0], p[0, 0, 0, 0, 0, 0], p[0, 0, 0, 0, 0, 0]]
          return pose_list
      end
      if length == 7:
          pose_list = [p[0, 0, 0, 0, 0, 0], p[0, 0, 0, 0, 0, 0], p[0, 0, 0, 0, 0, 0], p[0, 0, 0, 0, 0, 0], p[0, 0, 0, 0, 0, 0], p[0, 0, 0, 0, 0, 0], p[0, 0, 0, 0, 0, 0]]
          return pose_list
      end
      if length == 8:
          pose_list = [p[0, 0, 0, 0, 0, 0], p[0, 0, 0, 0, 0, 0], p[0, 0, 0, 0, 0, 0], p[0, 0, 0, 0, 0, 0], p[0, 0, 0, 0, 0, 0], p[0, 0, 0, 0, 0, 0], p[0, 0, 0, 0, 0, 0], p[0, 0, 0, 0, 0, 0]]
          return pose_list
      end
      if length == 9:
          pose_list = [p[0, 0, 0, 0, 0, 0], p[0, 0, 0, 0, 0, 0], p[0, 0, 0, 0, 0, 0], p[0, 0, 0, 0, 0, 0], p[0, 0, 0, 0, 0, 0], p[0, 0, 0, 0, 0, 0], p[0, 0, 0, 0, 0, 0], p[0, 0, 0, 0, 0, 0], p[0, 0, 0, 0, 0, 0]]
          return pose_list
      end
      if length > 9:
          popuptext = "Program is only capable of storing 9 pegs at once. You selected more than 9. "
          # infinite loop
          while 1==1:
              popup(popuptext, title="Too Many Pegs",blocking=True)
          end
      end
  end

  # this function calculates the poses required on the weldpath for a specific teach pose for peg center.
  # call this function for every peg you want to weld.
  def main_calculate_peg(pose1):
      # constants
      peg_width = 2.05 # inches
      fixture_height = 1.5 # inches
      cushout = 0.006 # 5mm # the cushion out from the wall
      cusharound = 0.004 # 5mm # the cushion around the sleeve.
      delz = fixture_height *25.4/1000 - cushout
      rad = peg_width *1/2 * 25.4/1000 + cusharound

      # calculate angles
      # rxryrz1 (for point 1 (back side of peg)
      # start with gun facing up, shield tip pointing in x+ direction
      # rotate about y axis (y-) 135 degrees.
      # thats it. (for the other ones, then rotate 90 degrees about z axis from this spot
      m0 = get_rotation_matrix_from_description("y", -1, 225 * pi / 180)
      rxryrz1 = convert_matrix_to_axang(m0)
      rx1 = rxryrz1[0]
      ry1 = rxryrz1[1]
      rz1 = rxryrz1[2]

      # rxryrz2
      # second rotation is 90 degrees about z- axis
      m1 = get_rotation_matrix_from_description("z", -1, 90 * pi / 180)
      m2 = multiply_matrix(m1, m0)
      rxryrz2 = convert_matrix_to_axang(m2)
      rx2 = rxryrz2[0]
      ry2 = rxryrz2[1]
      rz2 = rxryrz2[2]

      # rxryrz3
      # second rotation is 180 degrees about z- axis
      m1 = get_rotation_matrix_from_description("z", -1, 180 * pi / 180)
      m2 = multiply_matrix(m1, m0)
      rxryrz3 = convert_matrix_to_axang(m2)
      rx3 = rxryrz3[0]
      ry3 = rxryrz3[1]
      rz3 = rxryrz3[2]

      # rxryrz4
      # second rotation is 270 degrees about z- axis
      m1 = get_rotation_matrix_from_description("z", -1, 270 * pi / 180)
      m2 = multiply_matrix(m1, m0)
      rxryrz4 = convert_matrix_to_axang(m2)
      rx4 = rxryrz4[0]
      ry4 = rxryrz4[1]
      rz4 = rxryrz4[2]

      # get points
      # get lift column height based on z value
      # if z is between +1 feet and -1 feet then go to 750
      # if z is greater than +1 feet but less than +4 feet, then go to 880
      # if z is greater than +4 feet, then error
      # if z is less than -1 feet, then go to 750 mm above z.

      # scrap that. new rules
      # go to 750 mm above z.
      # if that result is above 880, then go to 880.
      # that will work until we get problems

      z0 = pose1[2] # the teach point's z value (taken when lift column = 0)
      lczn = z0 + .750 # lift column z needed
      if lczn > .880:
          lczn = .880
      end
      liftcolumnzneeded = lczn * 1000 # set the z position
      zposerel = z0 - lczn # z pose relative = the teach point's z value at the new lift column position.

      pcenterx = pose1[0]
      pcentery = pose1[1]

      #points
      p1x = pcenterx - rad
      p1y = pcentery
      p1z = zposerel - delz

      p2x = pcenterx
      p2y = pcentery + rad
      p2z = zposerel - delz

      p3x = pcenterx + rad
      p3y = pcentery
      p3z = zposerel - delz

      p4x = pcenterx
      p4y = pcentery - rad
      p4z = zposerel - delz

      point1 = p[p1x, p1y, p1z, rx1, ry1, rz1]
      point2 = p[p2x, p2y, p2z, rx2, ry2, rz2]
      point3 = p[p3x, p3y, p3z, rx3, ry3, rz3]
      point4 = p[p4x, p4y, p4z, rx4, ry4, rz4]

      ret = struct(point1=point1, point2=point2, point3=point3, point4=point4, liftcolumnzneeded=liftcolumnzneeded)
      return ret



  end
  $ 96 "leftchoice≔'Select Yes for a Left side weld, or select No for a Right Side weld.'"
  global leftchoice=request_boolean_from_primary_client("Select Yes for a Left side weld, or select No for a Right Side weld.")
  $ 97 "sidewallchoice≔'Is the sidewall 3/4 inch?'"
  global sidewallchoice=request_boolean_from_primary_client("Is the sidewall 3/4 inch?")
  $ 98 "If sidewallchoice"
  if (sidewallchoice):
    $ 99 "sidewall≔0.628"
    global sidewall=0.628
  else:
    $ 100 "Else" "noBreak"
    $ 101 "sidewall≔0.375"
    global sidewall=0.375
  end
  $ 102 "floorchoice≔'Is the floor 3/4 inch?'"
  global floorchoice=request_boolean_from_primary_client("Is the floor 3/4 inch?")
  $ 103 "If floorchoice"
  if (floorchoice):
    $ 104 "floorthick≔0.628"
    global floorthick=0.628
  else:
    $ 105 "Else" "noBreak"
    $ 106 "floorthick≔0.375"
    global floorthick=0.375
  end
  $ 107 "Set"
  set_tcp(p[-0.0095,-0.328,0.105,1.2092,-1.2092,1.2092])
  $ 108 "MoveJ"
  $ 109 "Waypoint_46" "breakAfter"
  movej(get_inverse_kin(Waypoint_46_p, qnear=Waypoint_46_q), a=1.3962634015954636, v=1.0471975511965976)
  $ 110 "Set"
  set_tcp(p[1.4000000000000001E-4,-0.01751,0.284,0.0,0.0,0.0])
  $ 111 "Test_Teach_Position()"
  Test_Teach_Position()
  $ 112 "Set"
  set_tcp(p[1.4000000000000001E-4,-0.01751,0.284,0.0,0.0,0.0])
  $ 113 "kill threadId_Thread_1"
  kill threadId_Thread_1
  $ 114 "Corner_Homing_45()"
  Corner_Homing_45()
  $ 115 "Set"
  set_tcp(p[-0.011699999999999999,-0.328,0.105,1.2092,-1.2092,1.2092])
  $ 120 "If leftchoice≟ True "
  if (leftchoice ==   True  ):
    $ 121 "pathturn≔main_calculate_left_extended(p11,p12,p21,p22,p3,p13,p23,sidewall,floorthick,tcp_pose_top)"
    global pathturn=main_calculate_left_extended(p11,p12,p21,p22,p3,p13,p23,sidewall,floorthick,tcp_pose_top)
    $ 122 "extrude_knife3()"
    extrude_knife3()
    $ 124 "move_path_3left()"
    move_path_3left()
  else:
    $ 125 "Else" "noBreak"
    $ 126 "pathturn≔main_calculate_right_extended(p11,p12,p21,p22,p3,p13,p23,sidewall,floorthick,tcp_pose_top)"
    global pathturn=main_calculate_right_extended(p11,p12,p21,p22,p3,p13,p23,sidewall,floorthick,tcp_pose_top)
    $ 127 "extrude_knife3()"
    extrude_knife3()
    $ 128 "move_path_3right()"
    move_path_3right()
  end
  $ 130 "MoveJ"
  $ 132 "Waypoint_20" "breakAfter"
  movej(get_inverse_kin(Waypoint_20_p, qnear=Waypoint_20_q), a=1.3962634015954636, v=1.0471975511965976)
  $ 133 "Home"
  movej([-3.266929759358355, -1.2139462677784536, 1.5878387874396154, 1.1069165929565088, -0.0023738326664366483, -1.7891447305770605], a=1.3962634015954636, v=1.0471975511965976)
end
